// TIA Portal V20 export
DATA_BLOCK "instLER_qrHistory_STK1Pos"   // DB306
// stored: InstanceOfName LER_qrHistory, InstanceOfType FB
"LER_qrHistory"
   // VAR_INPUT
   //    trigger : Bool;
   //    commonData : "LER_typeCommonData";
   //    qrData : "LER_typeQrData";
   // END_VAR
   // VAR_IN_OUT
   //    dataHistory : "LER_typeQrHistory";
   // END_VAR
   // VAR
   //    statDeleteData : "LER_typeQrHistory";
   //    statTrigger : Array[0..99] of Bool;
   //    statTonTimer { S7_SetPoint := 'True'} : Array[0..99] of TON_TIME;
   //    statComplete : Array[0..99] of Bool;
   // END_VAR
BEGIN
END_DATA_BLOCK
